FUNCTION_BLOCK FB_EventHandler
VAR_INPUT
	// PARENT / SETUP VARIABLES
	eParentID :  E_StateSourceID;
	sParentTrace : REFERENCE TO  T_MaxString;
	aErrorLog : REFERENCE TO ARRAY[1..dErrorLogMaxLength] OF ST_Event; 
	nErrorLogIndex : REFERENCE TO UINT;
	sLastParentInnerState : REFERENCE TO T_MaxString;
	sParentInnerState : REFERENCE TO T_MaxString;

	
	// CONTRROL FLAGS
	bAppendEvents : BOOL;
	bFrontEnd : BOOL;
	bLogState : BOOL;
	
	
	// LOCAL LOGGING INPUT VARS
	eNapID : E_Event := E_Event.NONE;
	nBeckhoffID : UDINT := 0;
	sTrace : T_MaxString;
	sErrorMessage : T_MaxString := '';
	sMessage : T_MaxString := '';
	
END_VAR

VAR
	bEvent : BOOL;
	stEvent : ARRAY[1..nArraySize] OF ST_Event; 
	nLocalErrorCount : UINT := 0; 
END_VAR


VAR CONSTANT
	nArraySize : UINT := 30;	// Local array size
	dErrorLogMaxLength : UINT := SystemConfig.MAIN_EVENT_LOG_MAX_LENGTH; // Global array size
END_VAR



// Add to local log queue if necessary
IF (eNapID <> E_Event.NONE) OR (nBeckhoffID <> 0) THEN
	UpdateParentTrace(); // Only update trace string when a new event comes in
	SaveEvent();
	AppendEvents();
END_IF


IF bAppendEvents THEN
	AppendEvents();				// Update main DB event array
END_IF


ResetEventVariables(); 		// Update internal variables

METHOD PRIVATE AppendEvents : BOOL
// Append events to the MAIN DB Array

WHILE nLocalErrorCount > 0 DO
	IF nErrorLogIndex < dErrorLogMaxLength THEN // TODO : Replace with global limit
		nErrorLogIndex := nErrorLogIndex + 1;
		aErrorLog[nErrorLogIndex] := GetEvent();
	END_IF
END_WHILE
END_METHOD

METHOD PRIVATE GetEvent : ST_Event
VAR
	Event : ST_Event;
	dCurrentErrorIndex : UINT := 1;
END_VAR

//Initialize default state object:	
Event.sEventTime := Datetime.GVL_TIME_STRING;
Event.eStateSourceID := TO_STRING(THIS^.eParentID);
Event.eNapEventID := TO_STRING(E_EventID.None);
Event.eBeckhoffErrorID := 0;
Event.eErrorSeverity := TO_STRING(E_ErrorSeverity.Event);
Event.sMessage := '';


IF nLocalErrorCount < 1 THEN
	// No errors to report
	GetEvent := Event;
	bEvent := FALSE;
	RETURN;
	
ELSE
	// Pop first index, shift remaining errors to front:
	Event := stEvent[1];
	
	// Check for severe error:
//	IF Event.eErrorSeverity = TO_STRING(E_ErrorSeverity.SevereError) THEN
//		bSevereError := TRUE;
//	END_IF
	
	WHILE dCurrentErrorIndex < nLocalErrorCount DO
		stEvent[dCurrentErrorIndex] := stEvent[dCurrentErrorIndex+1];
		dCurrentErrorIndex := dCurrentErrorIndex + 1;
	END_WHILE
	
	//Decrement error count to reflect the popped first index:
	nLocalErrorCount := nLocalErrorCount - 1;
	
	IF nLocalErrorCount < 1 THEN
		// We popped the last error:
		bEvent := FALSE;
	END_IF
	
END_IF

// Successfully popped error
GetEvent := Event;
END_METHOD

// Resets input variables that need to be reset each call to the FB_EventHandler
METHOD ResetEventVariables : BOOL
THIS^.eNapID := E_Event.NONE;
THIS^.nBeckhoffID := 0;

//THIS^.eTraceError := E_Event.NONE;
THIS^.sTrace := '';
THIS^.sMessage := '';

// Reset Flags
THIS^.bAppendEvents := FALSE;
THIS^.bFrontEnd := FALSE;
THIS^.bLogState := FALSE;
END_METHOD

METHOD PRIVATE SaveEvent : BOOL
VAR
	Event : ST_Event;
//	SeverityModulus : INT;
	dCurrentErrorIndex : UINT := 1;
	sStateTrans : T_MaxString;
END_VAR
// Build Temporary Event object:
Event.sEventTime := Datetime.GVL_TIME_STRING;
Event.eNapEventID := TO_STRING(THIS^.eNapID);
Event.eBeckhoffErrorID := THIS^.nBeckhoffID;
Event.bPassToFrontEnd := THIS^.bFrontEnd;
Event.eStateSourceID := TO_STRING(THIS^.eParentID);

IF THIS^.nBeckhoffID = 0 THEN
	// NAP Event/Error
	
//	SeverityModulus := (THIS^.eNapID MOD 500); // See E_ErrorID Enumeration for explanation
	
	IF eNapID < 1000 THEN
		Event.eErrorSeverity := TO_STRING(E_ErrorSeverity.Event);
	ELSIF eNapID < 2000 THEN
		Event.eErrorSeverity := TO_STRING(E_ErrorSeverity.Warning);
	ELSIF eNapID < 3000 THEN
		Event.eErrorSeverity := TO_STRING(E_ErrorSeverity.Error);
	ELSIF eNapID < 4000 THEN
		Event.eErrorSeverity := TO_STRING(E_ErrorSeverity.Info);
	ELSE
		Event.eErrorSeverity := TO_STRING(E_ErrorSeverity.Debug);	
	END_IF
	
	
ELSIF THIS^.eNapID = E_Event.NONE THEN
	// Beckhoff Error
	Event.eErrorSeverity := TO_STRING(E_ErrorSeverity.BeckhoffError);
ELSE
	// No error, should not get here.
	RETURN;
END_IF


// Build Event String
sStateTrans := CONCAT4('[',sLastParentInnerState,CONCAT('->',sParentInnerState),'] ');
IF sTrace = '' THEN
	// Only add message to event message
	Event.sMessage := CONCAT(sStateTrans,THIS^.sMessage);
ELSE
	// Add message AND trace to event message
	IF sMessage = '' THEN
		Event.sMessage := CONCAT(sStateTrans,THIS^.sParentTrace);
	ELSE
		Event.sMessage := CONCAT(sStateTrans,CONCAT(CONCAT(THIS^.sMessage,' >> '),THIS^.sParentTrace));
	END_IF

END_IF

IF nLocalErrorCount < nArraySize THEN
	// Array not filled, add new error to the back of queue:
	nLocalErrorCount := nLocalErrorCount + 1;
	stEvent[nLocalErrorCount] := Event;
	
ELSE
	// No increase in count if maximum size has already been reached
	WHILE dCurrentErrorIndex < nArraySize DO
		// Move all other indicies back 1 position, until we reach the front of queue:
		stEvent[dCurrentErrorIndex] := stEvent[dCurrentErrorIndex+1];	
		dCurrentErrorIndex := dCurrentErrorIndex + 1;
	END_WHILE
		// Save new error to the back:
		stEvent[nArraySize] := Event;
END_IF

// Redundant out of bounds error avoidance
IF nLocalErrorCount > nArraySize THEN
	nLocalErrorCount := nArraySize;
END_IF

THIS^.bEvent := TRUE;
//SaveEvent := TRUE;
END_METHOD

METHOD PUBLIC SaveState : BOOL


VAR_INPUT
	sLastState : T_MaxString := '';
	sNewState : T_MaxString := '';
	bOuter : BOOL;
END_VAR
VAR 
	Event : ST_Event;
	dCurrentErrorIndex : UINT := 1;
END_VAR
Event.sEventTime := Datetime.GVL_TIME_STRING;
Event.eBeckhoffErrorID := 0;
Event.bPassToFrontEnd := FALSE;
Event.eStateSourceID := TO_STRING(THIS^.eParentID);
Event.eErrorSeverity := TO_STRING(E_ErrorSeverity.Event);
IF bOuter THEN
	Event.sMessage := CONCAT(sLastState,CONCAT(' to ',sNewState));
	Event.eNapEventID := TO_STRING(E_Event.OUTER_STATE_CHANGE);
ELSE
	Event.sMessage := CONCAT(sLastState,CONCAT(' to ',sNewState));
	Event.eNapEventID := TO_STRING(E_Event.INNER_STATE_CHANGE);
END_IF


IF nLocalErrorCount < nArraySize THEN
	// Array not filled, add new error to the back of queue:
	nLocalErrorCount := nLocalErrorCount + 1;
	stEvent[nLocalErrorCount] := Event;
	
ELSE
	// No increase in count if maximum size has already been reached
	WHILE dCurrentErrorIndex < nArraySize DO
		// Move all other indicies back 1 position, until we reach the front of queue:
		stEvent[dCurrentErrorIndex] := stEvent[dCurrentErrorIndex+1];	
		dCurrentErrorIndex := dCurrentErrorIndex + 1;
	END_WHILE
		// Save new error to the back:
		stEvent[nArraySize] := Event;
END_IF

THIS^.bEvent := TRUE;
AppendEvents();
END_METHOD

// Sets the sParentTrace string appropriately, if inheiriting sTrace, it will append, otherwise it will start its own. 
// When a state machine issues an event with no sTrace specified, the sParentTrace is ignored while saving event.
METHOD UpdateParentTrace : BOOL
IF THIS^.sTrace = '' THEN
	// Build event trace
	IF THIS^.nBeckhoffID = 0 THEN
		// Append NAP Event to event trace
		THIS^.sParentTrace := CONCAT(CONCAT(TO_STRING(eParentID),'>>'),TO_STRING(THIS^.eNapID));
	ELSE
		// Append Beckhoff ID to event trace
		THIS^.sParentTrace := CONCAT(CONCAT(TO_STRING(eParentID),'>>'),CONCAT('Beckhoff ID: ',UDINT_TO_STRING(THIS^.nBeckhoffID)));
	END_IF
ELSE
	// Append child's event trace
	THIS^.sParentTrace := CONCAT(CONCAT(TO_STRING(THIS^.eParentID),'>>'),THIS^.sTrace);
END_IF
END_METHOD

END_FUNCTION_BLOCK

(* stored: Version 1.1.0.1, ProductVersion 3.1.4024.12
   POU FB_EventHandler: Id {ff0a1323-d03d-48f8-b1ca-30ec00608dfa}, SpecialFunc None
   Method AppendEvents: Id {4aec36a6-919e-4779-8edb-7ad0f86bd2c5}
   Method GetEvent: Id {7ddbc957-7b86-4369-9b01-11eee2c70257}
   Method ResetEventVariables: Id {b7212333-a690-4df6-b08b-d5c36341e0fc}
   Method SaveEvent: Id {bc2e4207-7f12-49fc-8338-dbb5792f5542}
   Method SaveState: Id {caefe455-73d8-47c5-b1cc-1d8c3dd05687}
   Method UpdateParentTrace: Id {bc830100-a566-4722-be2d-206500f3d50e} *)
